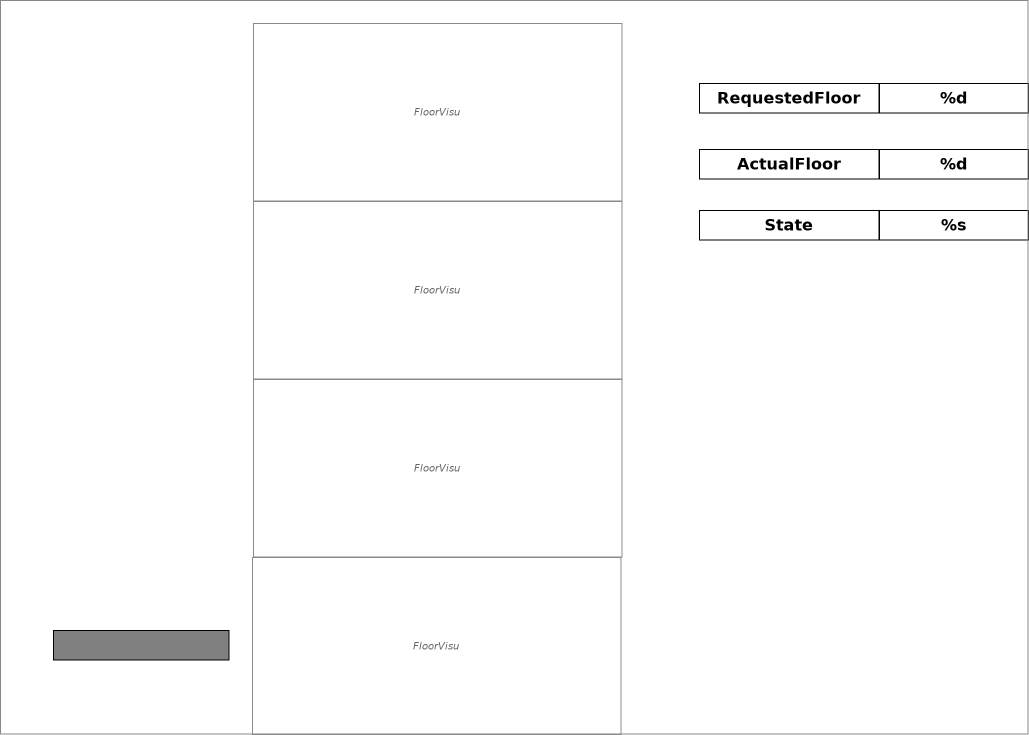
VISUALIZATION Visualization  // 1029x735
    Frame (252,557 369x178)
        shows FloorVisu(Callbt := Floors[1].Call, Low := Floors[1].Low, Mid := Floors[1].mid, High := Floors[1].High, name := BT_Text[1])
    Frame (253,379 369x178)
        shows FloorVisu(Callbt := Floors[2].Call, Low := Floors[2].Low, Mid := Floors[2].Mid, High := Floors[2].High, name := BT_Text[2])
    Frame (253,201 369x178)
        shows FloorVisu(Callbt := Floors[3].Call, Low := Floors[3].Low, Mid := Floors[3].Mid, High := Floors[3].High, name := BT_Text[3])
    Frame (253,23 369x178)
        shows FloorVisu(Callbt := Floors[4].Call, Low := Floors[4].Low, Mid := Floors[4].Mid, High := Floors[4].High, name := BT_Text[4])
    Rectangle (699,83 180x30), "RequestedFloor"
    Rectangle (699,149 180x30), "ActualFloor"
    Rectangle (879,83 150x30), "%d", text variable: RequestedFloor
    Rectangle (879,149 150x30), "%d", text variable: ActualFloor
    Rectangle (699,210 180x30), "State"
    Rectangle (879,210 150x30), "%s", text variable: MAIN.State
    Rectangle (53,630 176x30)
        p2738717112: Elevator_Y
END_VISUALIZATION

(* stored: Version 1.1.0.1, ProductVersion 3.1.4024.9
   Visu Visualization: Id {b58bdfba-9260-4a75-b9a7-c50b87f206da} *)
